{attribute 'qualified_only'}
VAR_GLOBAL
	location_lat	: LREAL; //{#lynus.ag#()}
	location_lon	: LREAL; //{#lynus.ag#()}
END_VAR

(* stored: Version 1.1.0.1, ProductVersion 3.1.4024.9
   GVL GVL: Id {4a18fc58-63da-4779-a177-12b25f261c54} *)
